FUNCTION_BLOCK S7_READ_CONTINUOUS
  {SET_ATTRIBUTE(OpcUa, DEVICE.SENSOR)}
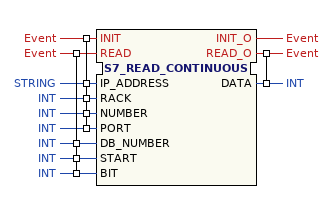
  EVENT_INPUT
    INIT WITH IP_ADDRESS, RACK, NUMBER, PORT;
    READ WITH DB_NUMBER, START, BIT;
  END_EVENT
  EVENT_OUTPUT
    INIT_O;
    READ_O WITH DATA;
  END_EVENT
  VAR_INPUT
    IP_ADDRESS : STRING; {SET_ATTRIBUTE(OpcUa, Constant.RUN)}
    RACK : INT; {SET_ATTRIBUTE(OpcUa, Constant.RUN)}
    NUMBER : INT; {SET_ATTRIBUTE(OpcUa, Constant.RUN)}
    PORT : INT; {SET_ATTRIBUTE(OpcUa, Constant.RUN)}
    DB_NUMBER : INT; {SET_ATTRIBUTE(OpcUa, Constant.RUN)}
    START : INT; {SET_ATTRIBUTE(OpcUa, Constant.RUN)}
    BIT : INT; {SET_ATTRIBUTE(OpcUa, Constant.RUN)}
  END_VAR
  VAR_OUTPUT
    DATA : INT; {SET_ATTRIBUTE(OpcUa, Variable.RUN)}
  END_VAR
END_FUNCTION_BLOCK
